// TwinCAT 3 PLC project HardwareSimulator
// ProgramVersion: 3.1.4024.0
// libraries:
//   Tc2_Standard, * (Beckhoff Automation GmbH)
//   Tc2_System, * (Beckhoff Automation GmbH)
//   Tc2_Utilities, * (Beckhoff Automation GmbH)
//   Tc3_Module, * (Beckhoff Automation GmbH)
//   VisuSymbols,3.5.10.0,System
// project tree:
//   / GlobalTextList.TcGTLO, PlcTask.TcTTO (not stored), Visualization Manager.TcVMO (not stored)
//   POUs/ MAIN.TcPOU, SIM_MOVITRAC_B2.TcPOU, SIM_ValveWithFB.TcPOU (not stored), SIM_ValveWithDoubleFB.TcPOU, SIM_MOVITRAC_B.TcPOU
//   VISUs/ Visualization.TcVIS (not stored)
// (motion and I/O tree: see PLC project cleanroomconnect)
// real-time tasks:
//   TASK PlcTask: cycle T#10ms, priority 20, ADS port 350
//   TASK PlcTask1: cycle T#10ms, priority 21, ADS port 351
//   TASK VISU_TASK: cycle T#200000us, priority 30, ADS port 352
// variable links:

// ---- POUs/MAIN.TcPOU
PROGRAM MAIN
VAR
	//EM Pallet Transport
	sim_MOVITRAC_B : SIM_MOVITRAC_B;
	//--sim_MOVITRAC_B2 : SIM_MOVITRAC_B2;
	simCentering : SIM_ValveWithDoubleFB;	

	//EM Docking Interface
	simDockingClampUpper : SIM_ValveWithDoubleFB;
	simDockingClampLower : SIM_ValveWithDoubleFB;
	simUnlockPinUpper : SIM_ValveWithFB;
	simUnlockPinLower : SIM_ValveWithFB;
	simDoorOpener : SIM_ValveWithFB;
	simDoorShutter : SIM_ValveWithFB;
	simDoorOpenerAlmostClosed AT %Q* : BOOL;
	tonDoorOpenerAlmosClosed : TON;
	
	simLiftActPosition AT %I* : LREAL;
	simLiftHomed AT %Q* : BOOL;
	simTransportUnitActPos AT %I* : LREAL;
	simTransportUnitHomed AT %Q* : BOOL;
	
	bInitDone : BOOL;
	simSafetyOK AT %Q* : BOOL;
	simPower400VacOK AT %Q* : BOOL;
	simPower230VacOK AT %Q* : BOOL;
	simPower230VacSocketsOK AT %Q* : BOOL;
	simPowerPotentialGroupOK AT %Q* : BOOL;
	simAirPressureOK AT %Q* : BOOL;
	simCabinetTemperatureOK AT %Q* : BOOL;
	
	
////{attribute 'TcLinkTo' := 'TIID^Device 1 (EtherCAT)^Term 1 (EK1100)^Term 2 (EL1004)^Channel 2^Input'}
(*	{attribute 'TcLinkTo' := 'TIPC^CleanroomConnect^CleanroomConnect Instance^PlcTask Outputs^GVL_Modules.g_emPalletConveyor.s_cmPalletConveyor.Q_bCmdReset'}
	I_bCmdReset AT %I* : BOOL;
	{attribute 'TcLinkTo' := 'TIPC^CleanroomConnect^CleanroomConnect Instance^PlcTask Outputs^GVL_Modules.g_emPalletConveyor.s_cmPalletConveyor.Q_bCmdEnable'}
	I_bCmdEnable AT %I* : BOOL;
	{attribute 'TcLinkTo' := 'TIPC^CleanroomConnect^CleanroomConnect Instance^PlcTask Outputs^GVL_Modules.g_emPalletConveyor.s_cmPalletConveyor.Q_bCmdStartCW'}
	I_bCmdStartCW AT %I* : BOOL;
	{attribute 'TcLinkTo' := 'TIPC^CleanroomConnect^CleanroomConnect Instance^PlcTask Outputs^GVL_Modules.g_emPalletConveyor.s_cmPalletConveyor.Q_bCmdStartCCW'}
	I_bCmdStartCCW AT %I* : BOOL;
	{attribute 'TcLinkTo' := 'TIPC^CleanroomConnect^CleanroomConnect Instance^PlcTask Inputs^GVL_Modules.g_emPalletConveyor.s_cmPalletConveyor.I_bStaReadyForOperation'}
	Q_bStaReadyForOperation AT %Q* : BOOL;
	{attribute 'TcLinkTo' := 'TIPC^CleanroomConnect^CleanroomConnect Instance^PlcTask Inputs^GVL_Modules.g_emPalletConveyor.s_cmPalletConveyor.I_bStaMotorIsRunning'}
	Q_bStaMotorIsRunning AT %Q* : BOOL;
*)	
END_VAR

IF NOT(bInitDone) THEN
	simSafetyOK := TRUE;
	simPower400VacOK := TRUE;
	simPower230VacOK := TRUE;
	simPower230VacSocketsOK := TRUE;
	simPowerPotentialGroupOK := TRUE;
	simAirPressureOK := TRUE;
	simCabinetTemperatureOK := TRUE;
	
	simDoorShutter.mForceOff();
	simDoorOpener.mForceOff();
	
	bInitDone := TRUE;
END_IF

//EM Pallet Conveyor
sim_MOVITRAC_B();
(*
sim_MOVITRAC_B2(
	i_ref_I_bCmdReset := I_bCmdReset, 
	i_ref_I_bCmdEnable := I_bCmdEnable, 
	i_ref_I_bCmdStartCW := I_bCmdStartCW, 
	i_ref_I_bCmdStartCCW := I_bCmdStartCCW, 
	i_ref_Q_bStaReadyForOperation := Q_bStaReadyForOperation, 
	i_ref_Q_bStaMotorIsRunning := Q_bStaMotorIsRunning);
*)
simCentering();

//EM Docking Interface
simDockingClampUpper();
simDockingClampLower();
simUnlockPinUpper();
simUnlockPinLower();
simDoorOpener();
simDoorShutter();

tonDoorOpenerAlmosClosed(IN := (simDoorOpener.q_bCmdValveOff OR simDoorOpener.q_bStaValveOff), PT := T#1S);
simDoorOpenerAlmostClosed := tonDoorOpenerAlmosClosed.Q; 

//IF (simLiftActPosition > 9999999000 AND simLiftActPosition < 10000000000 THEN
//simLiftHomed := TRUE;

//simLiftHomed := FALSE;

END_PROGRAM

// ---- POUs/SIM_MOVITRAC_B.TcPOU
FUNCTION_BLOCK SIM_MOVITRAC_B
VAR 
	// Outputs from PLC --> HW
	I_bCmdReset AT %I* : BOOL;
	I_bCmdEnable AT %I* : BOOL;
	I_bCmdStartCW AT %I* : BOOL;
	I_bCmdStartCCW AT %I* : BOOL;
	
	// Inputs from HW --> PLC
	Q_bStaReadyForOperation AT %Q* : BOOL;
	Q_bStaMotorIsRunning AT %Q* : BOOL;
	
	s_tonEnabled : TON;
	s_tonRunning : TON;
	s_tonStopped : TON;
	
	s_bError : BOOL := TRUE;	
END_VAR


s_tonEnabled(IN := (*I_bCmdEnable AND*) NOT(s_bError), PT := T#2S);
s_tonRunning(IN := s_tonEnabled.Q AND (I_bCmdStartCW OR I_bCmdStartCCW) , PT := T#2S);
s_tonStopped(IN := NOT(s_tonRunning.Q), PT := T#2S);

Q_bStaReadyForOperation := s_tonEnabled.Q;
Q_bStaMotorIsRunning := s_tonRunning.Q OR NOT(s_tonStopped.Q);

IF I_bCmdReset THEN
	s_bError := FALSE;
END_IF

END_FUNCTION_BLOCK

// ---- POUs/SIM_ValveWithDoubleFB.TcPOU
FUNCTION_BLOCK SIM_ValveWithDoubleFB
VAR 
	// Outputs from PLC --> HW
	I_bCmdValveOn AT %I* : BOOL;
	I_bCmdValveOff AT %I* : BOOL;
	
	// Inputs from HW --> PLC
	Q_bStaFeedbackOn AT %Q* : BOOL;
	Q_bStaFeedbackOff AT %Q* : BOOL;
	Q_bStaFeedbackOn2 AT %Q* : BOOL;
	Q_bStaFeedbackOff2 AT %Q* : BOOL;
	
	s_tonOn : TON;
	s_tonOff : TON;
	
END_VAR

VAR_OUTPUT
	q_bStaValveOn : BOOL;
	q_bStaValveOff : BOOL;
END_VAR


s_tonOn(IN := I_bCmdValveOn AND NOT(I_bCmdValveOff), PT := T#2S);

IF s_tonOn.Q THEN
	Q_bStaFeedbackOn := TRUE;
	Q_bStaFeedbackOn2 := TRUE;
ELSIF I_bCmdValveOff THEN
	Q_bStaFeedbackOn := FALSE;
	Q_bStaFeedbackOn2 := FALSE;
END_IF	
	
s_tonOff(IN := I_bCmdValveOff AND NOT(I_bCmdValveOn), PT := T#2S);

IF s_tonOff.Q THEN
	Q_bStaFeedbackOff := TRUE;
	Q_bStaFeedbackOff2 := TRUE;
ELSIF I_bCmdValveOn THEN
	Q_bStaFeedbackOff := FALSE;
	Q_bStaFeedbackOff2 := FALSE;
END_IF

q_bStaValveOn := Q_bStaFeedbackOn;
q_bStaValveOff := Q_bStaFeedbackOff;

END_FUNCTION_BLOCK

// ---- POUs/SIM_MOVITRAC_B2.TcPOU
FUNCTION_BLOCK SIM_MOVITRAC_B2
VAR_INPUT
	// Outputs from PLC --> HW
	i_ref_I_bCmdReset : REFERENCE TO BOOL;
	i_ref_I_bCmdEnable : REFERENCE TO BOOL;
	i_ref_I_bCmdStartCW : REFERENCE TO BOOL;
	i_ref_I_bCmdStartCCW : REFERENCE TO BOOL;
	
	// Inputs from HW --> PLC
	i_ref_Q_bStaReadyForOperation : REFERENCE TO BOOL;
	i_ref_Q_bStaMotorIsRunning : REFERENCE TO BOOL;
END_VAR
VAR 
	s_tonEnabled : TON;
	s_tonRunning : TON;
	s_tonStopped : TON;
	
	s_bError : BOOL := TRUE;	
END_VAR

s_tonEnabled(IN := (*I_bCmdEnable AND*) NOT(s_bError), PT := T#2S);
s_tonRunning(IN := s_tonEnabled.Q AND (i_ref_I_bCmdStartCW OR i_ref_I_bCmdStartCCW) , PT := T#2S);
s_tonStopped(IN := NOT(s_tonRunning.Q), PT := T#2S);

i_ref_Q_bStaReadyForOperation := s_tonEnabled.Q;
i_ref_Q_bStaMotorIsRunning := s_tonRunning.Q OR NOT(s_tonStopped.Q);

IF i_ref_I_bCmdReset THEN
	s_bError := FALSE;
END_IF

END_FUNCTION_BLOCK

// ---- GlobalTextList.TcGTLO
TEXTLIST GlobalTextList
  591 = 'dfgdfg'
  680 = 'Lower Clamps'
  564 = 'Upper Clamps'
END_TEXTLIST
